PROGRAM MAIN
VAR
	FirstEventInOurSturucture : ST_Events;
  	Boolean :BOOL := FALSE;
	eEventType : E_EventType := E_EventType.Alarm ;
	eEventSeverity : TcEventSeverity := TcEventSeverity.Error;
	eEventIdentity : UDINT := 777;
	eEventText : STRING(255) := 'BeCarefull';
	EventLogger : EvetLogger;
END_VAR


//FUpdateEventTimeStampedWithSystemTimeStamepd(FirstEventInOurSturucture);  
IF Boolean THEN 
	EventLogger.AddEvent(eEventType,eEventSeverity,eEventIdentity,eEventText);
END_IF

END_PROGRAM

(* stored: Version 1.1.0.1, ProductVersion 3.1.4024.12
   POU MAIN: Id {82d2561c-0b2b-45e9-b59f-2a3ce47a7c13}, SpecialFunc None *)
